(* CoDeSys 2.3.9.62 project: ComputeAngles.pro *)
(* Libraries: Standard.lib, Iecsfc.lib 8.11.10 11:37:48, SYSLIBCALLBACK.LIB *)

(* PLC configuration (modules and I/O channels)
K-Bus [K_Bus] node 0, in %IB0 out %QB0
Internal Digital I/O [InternalDigIO] node 1, in %IB512 out %QB512
  Internal Digital Inputs [Internal_DIN] node 0, in %IB512 out %QB512
    DIN1 AT %IX2300.0 [BOOLOnX_I] Internal Digital Input Bit 1
    DIN2 AT %IX2300.1 [BOOLOnX_I] Internal Digital Input Bit 2
  Internal Digital Outputs [Internal_DOUT] node 1, in %IB513 out %QB512
    DOUT1 AT %QX2300.0 [BOOLOnX_Q] Internal Digital Output Bit 1
    DOUT2 AT %QX2300.1 [BOOLOnX_Q] Internal Digital Output Bit 2
Fieldbus variables [FB_VARS] node 3, in %IB0 out %QB0
Flag variables [FLAG_VARS] node 4, in %IB0 out %QB0
Modbus-Master [MB_MASTER] node 5, in %IB0 out %QB0
*)

(* Task configuration *)
TASK NewTask (PRIORITY := 15);
	main();
END_TASK

(* POU main, ST *)
PROGRAM main
VAR

	ComputeAngles : ComputeAngles;

	roll : LREAL;
	pitch : LREAL;

	angle0 : LREAL;
	angle1 : LREAL;
	angle2 : LREAL;
	didBound : BOOL;

END_VAR
ComputeAngles.roll := roll;
ComputeAngles.pitch := pitch;

ComputeAngles();

angle0 := ComputeAngles.angle0;
angle1 := ComputeAngles.angle1;
angle2 := ComputeAngles.angle2;
didBound := ComputeAngles.didBound;
END_PROGRAM

(* POU ComputeAngles, ST *)
FUNCTION_BLOCK ComputeAngles
VAR_INPUT
	roll : LREAL;
	pitch : LREAL;
END_VAR
VAR_OUTPUT
	angle0 : LREAL;
	angle1 : LREAL;
	angle2 : LREAL;

	didBound : BOOL;
END_VAR
VAR
	l : LREAL := 1.75;
	delta : LREAL := 0.08;
	s0 : LREAL := 1.0;
	s1 : LREAL := 1.0;

	tmpVar0 : LREAL;
	tmpVar1 : LREAL;

	p0 : LREAL;
	p1 : LREAL;
	p2 : LREAL;
END_VAR
tmpVar0 := l / 2 * ATAN(roll / s1);
p1 :=delta + tmpVar0;
p0 := delta - tmpVar0;

tmpVar1 := (l * SQRT(3) / 2) * ATAN(pitch / s0) / 2.0;
p2 := delta - tmpVar1;

p0 := p0 + tmpVar1;
p1 := p1 + tmpVar1;

p0 := -1.0 * (p0 - delta) / delta;
p1 := -1.0 * (p1 - delta) / delta;
p2 := -1.0 * (p2 - delta) / delta;

didBound := FALSE;

IF (p0 > 1.0) THEN
	p0 := 1.0;
	didBound := TRUE;
ELSIF (p0 < -1.0) THEN
	p0 := -1.0;
	didBound := TRUE;
END_IF


IF (p1 > 1.0) THEN
	p1 := 1.0;
	didBound := TRUE;
ELSIF (p1 < -1.0) THEN
	p1 := -1.0;
	didBound := TRUE;
END_IF

IF (p2 > 1.0) THEN
	p2 := 1.0;
	didBound := TRUE;
ELSIF (p2 < -1.0) THEN
	p2 := -1.0;
	didBound := TRUE;
END_IF

angle0 := ACOS(p0);
angle1 := ACOS(p1);
angle2 := ACOS(p2);
END_FUNCTION_BLOCK
